KUKA KRL program: Fork_00_Milling_1.src

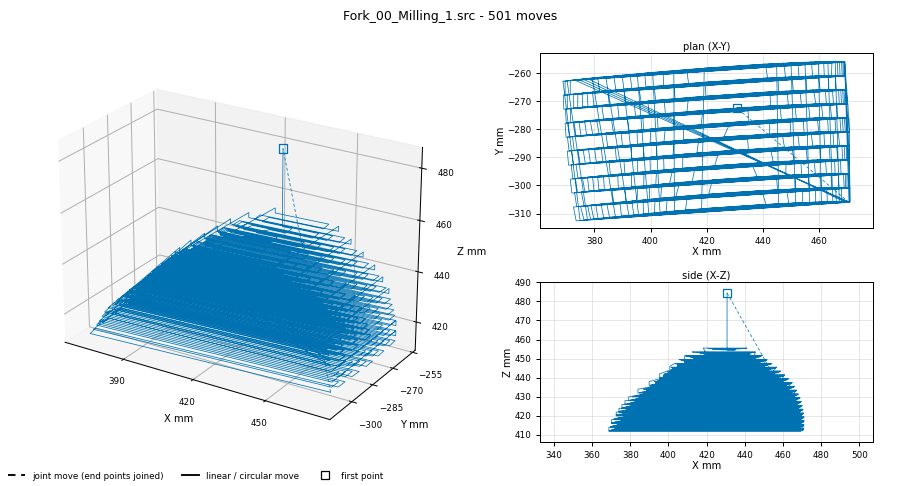
[picture p0: tool path of Fork_00_Milling_1.src, 501 of 503 moves have a stored position in this frame; points joined in program order, loops and branches not executed]
&ACCESS RVP
&REL 1
&PARAM TEMPLATE = C:\KRC\Roboter\Template\vorgabe
&PARAM EDITMASK = *
DEF milling_1 ( )


;FOLD INI
;FOLD BASISTECH INI
GLOBAL INTERRUPT DECL 3 WHEN $STOPMESS==TRUE DO IR_STOPM ( )
INTERRUPT ON 3
BAS (#INITMOV,0 )
;ENDFOLD (BASISTECH INI)
;ENDFOLD (INI)

;FOLD STARTPOSITION - BASE IS 0, TOOL IS 5, SPEED IS 15%, POSITION IS A1 5,A2 -90,A3 100,A4 5,A5 -10,A6 -5,E1 0,E2 0,E3 0,E4 0
$BWDSTART = FALSE
PDAT_ACT = {VEL 15,ACC 100,APO_DIST 50}
FDAT_ACT = {TOOL_NO 5,BASE_NO 0,IPO_FRAME #BASE}
BAS (#PTP_PARAMS,15)
PTP  {A1 5,A2 -90,A3 100,A4 5,A5 -10,A6 -5,E1 0,E2 0,E3 0,E4 0}
;ENDFOLD

;FOLD LIN SPEED IS 0.1 m/sec, INTERPOLATION SETTINGS IN FOLD
$VEL.CP=0.1
$ADVANCE=3
;ENDFOLD

BAS(#VEL_PTP,2)
PTP {X 430.72, Y -272.354, Z 484.436, A 0, B 90, C 0, E1 0, E2 0, E3 0, E4 0, S 'B010'}
$VEL.CP=0.005
LIN {X 430.72, Y -272.354, Z 454.436, A 0, B 90, C 0, E1 0, E2 0, E3 0, E4 0}
LIN {X 434.594, Y -272.091, Z 454.436, A 0, B 90, C 0, E1 0, E2 0, E3 0, E4 0}
LIN {X 435.068, Y -277.068, Z 454.593, A 0, B 90, C 0, E1 0, E2 0, E3 0, E4 0}
LIN {X 428.455, Y -277.517, Z 454.593, A 0, B 90, C 0, E1 0, E2 0, E3 0, E4 0}
LIN {X 426.127, Y -282.684, Z 454.749, A 0, B 90, C 0, E1 0, E2 0, E3 0, E4 0}
LIN {X 434.47, Y -282.118, Z 454.75, A 0, B 90, C 0, E1 0, E2 0, E3 0, E4 0}
LIN {X 434.889, Y -287.099, Z 454.906, A 0, B 90, C 0, E1 0, E2 0, E3 0, E4 0}
LIN {X 424.389, Y -287.811, Z 454.906, A 0, B 90, C 0, E1 0, E2 0, E3 0, E4 0}
LIN {X 422.898, Y -292.921, Z 455.063, A 0, B 90, C 0, E1 0, E2 0, E3 0, E4 0}
LIN {X 435.962, Y -292.035, Z 455.063, A 0, B 90, C 0, E1 0, E2 0, E3 0, E4 0}
LIN {X 437.991, Y -296.906, Z 455.22, A 0, B 90, C 0, E1 0, E2 0, E3 0, E4 0}
LIN {X 422.043, Y -297.989, Z 455.22, A 0, B 90, C 0, E1 0, E2 0, E3 0, E4 0}
LIN {X 420.746, Y -303.086, Z 455.376, A 0, B 90, C 0, E1 0, E2 0, E3 0, E4 0}
LIN {X 439.68, Y -301.801, Z 455.377, A 0, B 90, C 0, E1 0, E2 0, E3 0, E4 0}
LIN {X 441.144, Y -306.71, Z 455.534, A 0, B 90, C 0, E1 0, E2 0, E3 0, E4 0}
LIN {X 418.215, Y -308.266, Z 455.533, A 0, B 90, C 0, E1 0, E2 0, E3 0, E4 0}
LIN {X 419.146, Y -258.113, Z 453.965, A 0, B 90, C 0, E1 0, E2 0, E3 0, E4 0}
LIN {X 419.15, Y -258.175, Z 451.966, A 0, B 90, C 0, E1 0, E2 0, E3 0, E4 0}
LIN {X 440.969, Y -256.694, Z 451.966, A 0, B 90, C 0, E1 0, E2 0, E3 0, E4 0}
LIN {X 441.697, Y -261.654, Z 452.123, A 0, B 90, C 0, E1 0, E2 0, E3 0, E4 0}
LIN {X 419.492, Y -263.161, Z 452.123, A 0, B 90, C 0, E1 0, E2 0, E3 0, E4 0}
LIN {X 419.733, Y -268.154, Z 452.279, A 0, B 90, C 0, E1 0, E2 0, E3 0, E4 0}
LIN {X 442.505, Y -266.608, Z 452.28, A 0, B 90, C 0, E1 0, E2 0, E3 0, E4 0}
LIN {X 442.855, Y -271.594, Z 452.437, A 0, B 90, C 0, E1 0, E2 0, E3 0, E4 0}
LIN {X 418.625, Y -273.238, Z 452.436, A 0, B 90, C 0, E1 0, E2 0, E3 0, E4 0}
LIN {X 418.028, Y -278.288, Z 452.593, A 0, B 90, C 0, E1 0, E2 0, E3 0, E4 0}
LIN {X 442.441, Y -276.631, Z 452.594, A 0, B 90, C 0, E1 0, E2 0, E3 0, E4 0}
LIN {X 442.487, Y -281.637, Z 452.75, A 0, B 90, C 0, E1 0, E2 0, E3 0, E4 0}
LIN {X 417.259, Y -283.349, Z 452.75, A 0, B 90, C 0, E1 0, E2 0, E3 0, E4 0}
LIN {X 416.509, Y -288.409, Z 452.906, A 0, B 90, C 0, E1 0, E2 0, E3 0, E4 0}
LIN {X 442.672, Y -286.633, Z 452.907, A 0, B 90, C 0, E1 0, E2 0, E3 0, E4 0}
LIN {X 443.761, Y -291.568, Z 453.064, A 0, B 90, C 0, E1 0, E2 0, E3 0, E4 0}
LIN {X 415.871, Y -293.461, Z 453.063, A 0, B 90, C 0, E1 0, E2 0, E3 0, E4 0}
LIN {X 414.841, Y -298.54, Z 453.22, A 0, B 90, C 0, E1 0, E2 0, E3 0, E4 0}
LIN {X 444.838, Y -296.504, Z 453.221, A 0, B 90, C 0, E1 0, E2 0, E3 0, E4 0}
LIN {X 445.27, Y -301.484, Z 453.378, A 0, B 90, C 0, E1 0, E2 0, E3 0, E4 0}
LIN {X 413.14, Y -303.665, Z 453.377, A 0, B 90, C 0, E1 0, E2 0, E3 0, E4 0}
LIN {X 412.448, Y -308.721, Z 453.534, A 0, B 90, C 0, E1 0, E2 0, E3 0, E4 0}
LIN {X 445.669, Y -306.466, Z 453.534, A 0, B 90, C 0, E1 0, E2 0, E3 0, E4 0}
LIN {X 444.959, Y -256.424, Z 451.967, A 0, B 90, C 0, E1 0, E2 0, E3 0, E4 0}
LIN {X 444.964, Y -256.486, Z 449.968, A 0, B 90, C 0, E1 0, E2 0, E3 0, E4 0}
LIN {X 412.911, Y -258.662, Z 449.967, A 0, B 90, C 0, E1 0, E2 0, E3 0, E4 0}
LIN {X 413.546, Y -263.628, Z 450.124, A 0, B 90, C 0, E1 0, E2 0, E3 0, E4 0}
LIN {X 445.401, Y -261.466, Z 450.124, A 0, B 90, C 0, E1 0, E2 0, E3 0, E4 0}
LIN {X 445.696, Y -266.455, Z 450.281, A 0, B 90, C 0, E1 0, E2 0, E3 0, E4 0}
LIN {X 413.503, Y -268.64, Z 450.281, A 0, B 90, C 0, E1 0, E2 0, E3 0, E4 0}
LIN {X 413.007, Y -273.682, Z 450.437, A 0, B 90, C 0, E1 0, E2 0, E3 0, E4 0}
LIN {X 446.106, Y -271.436, Z 450.438, A 0, B 90, C 0, E1 0, E2 0, E3 0, E4 0}
LIN {X 446.657, Y -276.407, Z 450.595, A 0, B 90, C 0, E1 0, E2 0, E3 0, E4 0}
LIN {X 411.832, Y -278.771, Z 450.594, A 0, B 90, C 0, E1 0, E2 0, E3 0, E4 0}
LIN {X 411.67, Y -283.791, Z 450.751, A 0, B 90, C 0, E1 0, E2 0, E3 0, E4 0}
LIN {X 446.887, Y -281.401, Z 450.752, A 0, B 90, C 0, E1 0, E2 0, E3 0, E4 0}
LIN {X 447.736, Y -286.352, Z 450.908, A 0, B 90, C 0, E1 0, E2 0, E3 0, E4 0}
LIN {X 411.519, Y -288.811, Z 450.908, A 0, B 90, C 0, E1 0, E2 0, E3 0, E4 0}
LIN {X 411.454, Y -293.824, Z 451.064, A 0, B 90, C 0, E1 0, E2 0, E3 0, E4 0}
LIN {X 448.317, Y -291.322, Z 451.065, A 0, B 90, C 0, E1 0, E2 0, E3 0, E4 0}
LIN {X 448.215, Y -296.338, Z 451.222, A 0, B 90, C 0, E1 0, E2 0, E3 0, E4 0}
LIN {X 410.374, Y -298.906, Z 451.221, A 0, B 90, C 0, E1 0, E2 0, E3 0, E4 0}
LIN {X 409.012, Y -304.008, Z 451.378, A 0, B 90, C 0, E1 0, E2 0, E3 0, E4 0}
LIN {X 448.504, Y -301.327, Z 451.379, A 0, B 90, C 0, E1 0, E2 0, E3 0, E4 0}
LIN {X 449.256, Y -306.285, Z 451.536, A 0, B 90, C 0, E1 0, E2 0, E3 0, E4 0}
LIN {X 408.508, Y -309.051, Z 451.535, A 0, B 90, C 0, E1 0, E2 0, E3 0, E4 0}
LIN {X 408.295, Y -258.975, Z 449.967, A 0, B 90, C 0, E1 0, E2 0, E3 0, E4 0}
LIN {X 408.299, Y -259.038, Z 447.968, A 0, B 90, C 0, E1 0, E2 0, E3 0, E4 0}
LIN {X 447.536, Y -256.374, Z 447.969, A 0, B 90, C 0, E1 0, E2 0, E3 0, E4 0}
LIN {X 448.106, Y -261.345, Z 448.126, A 0, B 90, C 0, E1 0, E2 0, E3 0, E4 0}
LIN {X 408.404, Y -264.04, Z 448.125, A 0, B 90, C 0, E1 0, E2 0, E3 0, E4 0}
LIN {X 408.727, Y -269.027, Z 448.281, A 0, B 90, C 0, E1 0, E2 0, E3 0, E4 0}
LIN {X 448.61, Y -266.32, Z 448.282, A 0, B 90, C 0, E1 0, E2 0, E3 0, E4 0}
LIN {X 449.134, Y -271.293, Z 448.439, A 0, B 90, C 0, E1 0, E2 0, E3 0, E4 0}
LIN {X 408.355, Y -274.061, Z 448.438, A 0, B 90, C 0, E1 0, E2 0, E3 0, E4 0}
LIN {X 408.359, Y -279.07, Z 448.595, A 0, B 90, C 0, E1 0, E2 0, E3 0, E4 0}
LIN {X 449.68, Y -276.265, Z 448.596, A 0, B 90, C 0, E1 0, E2 0, E3 0, E4 0}
LIN {X 450.001, Y -281.252, Z 448.753, A 0, B 90, C 0, E1 0, E2 0, E3 0, E4 0}
LIN {X 408.293, Y -284.083, Z 448.752, A 0, B 90, C 0, E1 0, E2 0, E3 0, E4 0}
LIN {X 408.039, Y -289.11, Z 448.909, A 0, B 90, C 0, E1 0, E2 0, E3 0, E4 0}
LIN {X 450.372, Y -286.236, Z 448.909, A 0, B 90, C 0, E1 0, E2 0, E3 0, E4 0}
LIN {X 451.141, Y -291.193, Z 449.066, A 0, B 90, C 0, E1 0, E2 0, E3 0, E4 0}
LIN {X 407.934, Y -294.126, Z 449.065, A 0, B 90, C 0, E1 0, E2 0, E3 0, E4 0}
LIN {X 406.788, Y -299.213, Z 449.222, A 0, B 90, C 0, E1 0, E2 0, E3 0, E4 0}
LIN {X 451.562, Y -296.174, Z 449.223, A 0, B 90, C 0, E1 0, E2 0, E3 0, E4 0}
LIN {X 451.599, Y -301.18, Z 449.38, A 0, B 90, C 0, E1 0, E2 0, E3 0, E4 0}
LIN {X 405.979, Y -304.277, Z 449.379, A 0, B 90, C 0, E1 0, E2 0, E3 0, E4 0}
LIN {X 405.553, Y -309.315, Z 449.536, A 0, B 90, C 0, E1 0, E2 0, E3 0, E4 0}
LIN {X 451.726, Y -306.18, Z 449.537, A 0, B 90, C 0, E1 0, E2 0, E3 0, E4 0}
LIN {X 450.067, Y -256.203, Z 447.969, A 0, B 90, C 0, E1 0, E2 0, E3 0, E4 0}
LIN {X 450.071, Y -256.265, Z 445.97, A 0, B 90, C 0, E1 0, E2 0, E3 0, E4 0}
LIN {X 404.497, Y -259.359, Z 445.969, A 0, B 90, C 0, E1 0, E2 0, E3 0, E4 0}
LIN {X 404.613, Y -264.36, Z 446.125, A 0, B 90, C 0, E1 0, E2 0, E3 0, E4 0}
LIN {X 450.414, Y -261.251, Z 446.127, A 0, B 90, C 0, E1 0, E2 0, E3 0, E4 0}
LIN {X 450.904, Y -266.227, Z 446.283, A 0, B 90, C 0, E1 0, E2 0, E3 0, E4 0}
LIN {X 404.855, Y -269.352, Z 446.282, A 0, B 90, C 0, E1 0, E2 0, E3 0, E4 0}
LIN {X 405.282, Y -274.333, Z 446.439, A 0, B 90, C 0, E1 0, E2 0, E3 0, E4 0}
LIN {X 451.426, Y -271.2, Z 446.44, A 0, B 90, C 0, E1 0, E2 0, E3 0, E4 0}
LIN {X 451.972, Y -276.172, Z 446.597, A 0, B 90, C 0, E1 0, E2 0, E3 0, E4 0}
LIN {X 405.292, Y -279.341, Z 446.596, A 0, B 90, C 0, E1 0, E2 0, E3 0, E4 0}
LIN {X 404.784, Y -284.384, Z 446.753, A 0, B 90, C 0, E1 0, E2 0, E3 0, E4 0}
LIN {X 452.413, Y -281.151, Z 446.754, A 0, B 90, C 0, E1 0, E2 0, E3 0, E4 0}
LIN {X 453.043, Y -286.118, Z 446.911, A 0, B 90, C 0, E1 0, E2 0, E3 0, E4 0}
LIN {X 404.634, Y -289.404, Z 446.909, A 0, B 90, C 0, E1 0, E2 0, E3 0, E4 0}
LIN {X 404.807, Y -294.401, Z 447.066, A 0, B 90, C 0, E1 0, E2 0, E3 0, E4 0}
LIN {X 453.573, Y -291.091, Z 447.067, A 0, B 90, C 0, E1 0, E2 0, E3 0, E4 0}
LIN {X 453.857, Y -296.081, Z 447.224, A 0, B 90, C 0, E1 0, E2 0, E3 0, E4 0}
LIN {X 404.012, Y -299.464, Z 447.223, A 0, B 90, C 0, E1 0, E2 0, E3 0, E4 0}
LIN {X 403.621, Y -304.499, Z 447.38, A 0, B 90, C 0, E1 0, E2 0, E3 0, E4 0}
LIN {X 454.257, Y -301.063, Z 447.381, A 0, B 90, C 0, E1 0, E2 0, E3 0, E4 0}
LIN {X 454.181, Y -306.077, Z 447.538, A 0, B 90, C 0, E1 0, E2 0, E3 0, E4 0}
LIN {X 403.378, Y -309.525, Z 447.536, A 0, B 90, C 0, E1 0, E2 0, E3 0, E4 0}
LIN {X 400.738, Y -259.614, Z 445.969, A 0, B 90, C 0, E1 0, E2 0, E3 0, E4 0}
LIN {X 400.743, Y -259.676, Z 443.969, A 0, B 90, C 0, E1 0, E2 0, E3 0, E4 0}
LIN {X 452.557, Y -256.159, Z 443.971, A 0, B 90, C 0, E1 0, E2 0, E3 0, E4 0}
LIN {X 452.9, Y -261.145, Z 444.127, A 0, B 90, C 0, E1 0, E2 0, E3 0, E4 0}
LIN {X 401.269, Y -264.65, Z 444.126, A 0, B 90, C 0, E1 0, E2 0, E3 0, E4 0}
LIN {X 401.82, Y -269.621, Z 444.283, A 0, B 90, C 0, E1 0, E2 0, E3 0, E4 0}
LIN {X 453.243, Y -266.131, Z 444.284, A 0, B 90, C 0, E1 0, E2 0, E3 0, E4 0}
LIN {X 453.757, Y -271.105, Z 444.441, A 0, B 90, C 0, E1 0, E2 0, E3 0, E4 0}
LIN {X 402.363, Y -274.594, Z 444.44, A 0, B 90, C 0, E1 0, E2 0, E3 0, E4 0}
LIN {X 402.668, Y -279.582, Z 444.597, A 0, B 90, C 0, E1 0, E2 0, E3 0, E4 0}
LIN {X 454.371, Y -276.072, Z 444.598, A 0, B 90, C 0, E1 0, E2 0, E3 0, E4 0}
LIN {X 454.728, Y -281.057, Z 444.755, A 0, B 90, C 0, E1 0, E2 0, E3 0, E4 0}
LIN {X 402.155, Y -284.626, Z 444.753, A 0, B 90, C 0, E1 0, E2 0, E3 0, E4 0}
LIN {X 402.095, Y -289.639, Z 444.91, A 0, B 90, C 0, E1 0, E2 0, E3 0, E4 0}
LIN {X 455.371, Y -286.023, Z 444.911, A 0, B 90, C 0, E1 0, E2 0, E3 0, E4 0}
LIN {X 455.856, Y -290.999, Z 445.068, A 0, B 90, C 0, E1 0, E2 0, E3 0, E4 0}
LIN {X 402.122, Y -294.646, Z 445.067, A 0, B 90, C 0, E1 0, E2 0, E3 0, E4 0}
LIN {X 401.877, Y -299.672, Z 445.224, A 0, B 90, C 0, E1 0, E2 0, E3 0, E4 0}
LIN {X 456.278, Y -295.979, Z 445.225, A 0, B 90, C 0, E1 0, E2 0, E3 0, E4 0}
LIN {X 456.604, Y -300.966, Z 445.382, A 0, B 90, C 0, E1 0, E2 0, E3 0, E4 0}
LIN {X 401.627, Y -304.698, Z 445.381, A 0, B 90, C 0, E1 0, E2 0, E3 0, E4 0}
LIN {X 401.381, Y -309.723, Z 445.537, A 0, B 90, C 0, E1 0, E2 0, E3 0, E4 0}
LIN {X 456.676, Y -305.97, Z 445.539, A 0, B 90, C 0, E1 0, E2 0, E3 0, E4 0}
LIN {X 455.057, Y -255.99, Z 443.971, A 0, B 90, C 0, E1 0, E2 0, E3 0, E4 0}
LIN {X 455.062, Y -256.052, Z 441.972, A 0, B 90, C 0, E1 0, E2 0, E3 0, E4 0}
LIN {X 397.907, Y -259.932, Z 441.97, A 0, B 90, C 0, E1 0, E2 0, E3 0, E4 0}
LIN {X 398.366, Y -264.91, Z 442.127, A 0, B 90, C 0, E1 0, E2 0, E3 0, E4 0}
LIN {X 455.403, Y -261.038, Z 442.128, A 0, B 90, C 0, E1 0, E2 0, E3 0, E4 0}
LIN {X 455.72, Y -266.026, Z 442.285, A 0, B 90, C 0, E1 0, E2 0, E3 0, E4 0}
LIN {X 398.99, Y -269.876, Z 442.284, A 0, B 90, C 0, E1 0, E2 0, E3 0, E4 0}
LIN {X 399.564, Y -274.846, Z 442.441, A 0, B 90, C 0, E1 0, E2 0, E3 0, E4 0}
LIN {X 456.275, Y -270.997, Z 442.442, A 0, B 90, C 0, E1 0, E2 0, E3 0, E4 0}
LIN {X 456.818, Y -275.969, Z 442.599, A 0, B 90, C 0, E1 0, E2 0, E3 0, E4 0}
LIN {X 400.065, Y -279.821, Z 442.597, A 0, B 90, C 0, E1 0, E2 0, E3 0, E4 0}
LIN {X 399.84, Y -284.846, Z 442.754, A 0, B 90, C 0, E1 0, E2 0, E3 0, E4 0}
LIN {X 457.204, Y -280.952, Z 442.756, A 0, B 90, C 0, E1 0, E2 0, E3 0, E4 0}
LIN {X 457.852, Y -285.917, Z 442.912, A 0, B 90, C 0, E1 0, E2 0, E3 0, E4 0}
LIN {X 399.811, Y -289.857, Z 442.911, A 0, B 90, C 0, E1 0, E2 0, E3 0, E4 0}
LIN {X 399.908, Y -294.859, Z 443.068, A 0, B 90, C 0, E1 0, E2 0, E3 0, E4 0}
LIN {X 458.35, Y -290.892, Z 443.069, A 0, B 90, C 0, E1 0, E2 0, E3 0, E4 0}
LIN {X 458.732, Y -295.875, Z 443.226, A 0, B 90, C 0, E1 0, E2 0, E3 0, E4 0}
LIN {X 399.751, Y -299.879, Z 443.225, A 0, B 90, C 0, E1 0, E2 0, E3 0, E4 0}
LIN {X 399.552, Y -304.901, Z 443.381, A 0, B 90, C 0, E1 0, E2 0, E3 0, E4 0}
LIN {X 458.809, Y -300.879, Z 443.383, A 0, B 90, C 0, E1 0, E2 0, E3 0, E4 0}
LIN {X 458.885, Y -305.883, Z 443.54, A 0, B 90, C 0, E1 0, E2 0, E3 0, E4 0}
LIN {X 399.354, Y -309.924, Z 443.538, A 0, B 90, C 0, E1 0, E2 0, E3 0, E4 0}
LIN {X 395.258, Y -260.112, Z 441.97, A 0, B 90, C 0, E1 0, E2 0, E3 0, E4 0}
LIN {X 395.262, Y -260.174, Z 439.971, A 0, B 90, C 0, E1 0, E2 0, E3 0, E4 0}
LIN {X 457.344, Y -255.96, Z 439.972, A 0, B 90, C 0, E1 0, E2 0, E3 0, E4 0}
LIN {X 457.776, Y -260.94, Z 440.129, A 0, B 90, C 0, E1 0, E2 0, E3 0, E4 0}
LIN {X 395.84, Y -265.144, Z 440.128, A 0, B 90, C 0, E1 0, E2 0, E3 0, E4 0}
LIN {X 396.614, Y -270.1, Z 440.285, A 0, B 90, C 0, E1 0, E2 0, E3 0, E4 0}
LIN {X 458.111, Y -265.926, Z 440.286, A 0, B 90, C 0, E1 0, E2 0, E3 0, E4 0}
LIN {X 458.91, Y -270.881, Z 440.443, A 0, B 90, C 0, E1 0, E2 0, E3 0, E4 0}
LIN {X 397.252, Y -275.066, Z 440.441, A 0, B 90, C 0, E1 0, E2 0, E3 0, E4 0}
LIN {X 397.475, Y -280.06, Z 440.598, A 0, B 90, C 0, E1 0, E2 0, E3 0, E4 0}
LIN {X 459.417, Y -275.856, Z 440.6, A 0, B 90, C 0, E1 0, E2 0, E3 0, E4 0}
LIN {X 459.985, Y -280.826, Z 440.756, A 0, B 90, C 0, E1 0, E2 0, E3 0, E4 0}
LIN {X 397.521, Y -285.066, Z 440.755, A 0, B 90, C 0, E1 0, E2 0, E3 0, E4 0}
LIN {X 397.583, Y -290.071, Z 440.912, A 0, B 90, C 0, E1 0, E2 0, E3 0, E4 0}
LIN {X 460.359, Y -285.81, Z 440.913, A 0, B 90, C 0, E1 0, E2 0, E3 0, E4 0}
LIN {X 460.544, Y -290.806, Z 441.07, A 0, B 90, C 0, E1 0, E2 0, E3 0, E4 0}
LIN {X 397.674, Y -295.074, Z 441.069, A 0, B 90, C 0, E1 0, E2 0, E3 0, E4 0}
LIN {X 397.572, Y -300.09, Z 441.225, A 0, B 90, C 0, E1 0, E2 0, E3 0, E4 0}
LIN {X 460.729, Y -295.803, Z 441.227, A 0, B 90, C 0, E1 0, E2 0, E3 0, E4 0}
LIN {X 460.84, Y -300.804, Z 441.384, A 0, B 90, C 0, E1 0, E2 0, E3 0, E4 0}
LIN {X 397.374, Y -305.112, Z 441.382, A 0, B 90, C 0, E1 0, E2 0, E3 0, E4 0}
LIN {X 397.441, Y -310.117, Z 441.539, A 0, B 90, C 0, E1 0, E2 0, E3 0, E4 0}
LIN {X 460.897, Y -305.809, Z 441.54, A 0, B 90, C 0, E1 0, E2 0, E3 0, E4 0}
LIN {X 459.838, Y -255.791, Z 439.972, A 0, B 90, C 0, E1 0, E2 0, E3 0, E4 0}
LIN {X 459.842, Y -255.853, Z 437.973, A 0, B 90, C 0, E1 0, E2 0, E3 0, E4 0}
LIN {X 392.711, Y -260.41, Z 437.972, A 0, B 90, C 0, E1 0, E2 0, E3 0, E4 0}
LIN {X 393.304, Y -265.379, Z 438.129, A 0, B 90, C 0, E1 0, E2 0, E3 0, E4 0}
LIN {X 459.891, Y -260.859, Z 438.13, A 0, B 90, C 0, E1 0, E2 0, E3 0, E4 0}
LIN {X 460.475, Y -265.829, Z 438.287, A 0, B 90, C 0, E1 0, E2 0, E3 0, E4 0}
LIN {X 394.093, Y -270.334, Z 438.285, A 0, B 90, C 0, E1 0, E2 0, E3 0, E4 0}
LIN {X 394.69, Y -275.303, Z 438.442, A 0, B 90, C 0, E1 0, E2 0, E3 0, E4 0}
LIN {X 460.924, Y -270.807, Z 438.444, A 0, B 90, C 0, E1 0, E2 0, E3 0, E4 0}
LIN {X 461.398, Y -275.784, Z 438.601, A 0, B 90, C 0, E1 0, E2 0, E3 0, E4 0}
LIN {X 395.156, Y -280.28, Z 438.599, A 0, B 90, C 0, E1 0, E2 0, E3 0, E4 0}
LIN {X 395.334, Y -285.277, Z 438.756, A 0, B 90, C 0, E1 0, E2 0, E3 0, E4 0}
LIN {X 461.793, Y -280.766, Z 438.757, A 0, B 90, C 0, E1 0, E2 0, E3 0, E4 0}
LIN {X 462.025, Y -285.76, Z 438.914, A 0, B 90, C 0, E1 0, E2 0, E3 0, E4 0}
LIN {X 395.356, Y -290.285, Z 438.913, A 0, B 90, C 0, E1 0, E2 0, E3 0, E4 0}
LIN {X 395.431, Y -295.289, Z 439.069, A 0, B 90, C 0, E1 0, E2 0, E3 0, E4 0}
LIN {X 462.369, Y -290.745, Z 439.071, A 0, B 90, C 0, E1 0, E2 0, E3 0, E4 0}
LIN {X 462.701, Y -295.732, Z 439.228, A 0, B 90, C 0, E1 0, E2 0, E3 0, E4 0}
LIN {X 395.383, Y -300.301, Z 439.226, A 0, B 90, C 0, E1 0, E2 0, E3 0, E4 0}
LIN {X 395.185, Y -305.324, Z 439.383, A 0, B 90, C 0, E1 0, E2 0, E3 0, E4 0}
LIN {X 462.857, Y -300.73, Z 439.384, A 0, B 90, C 0, E1 0, E2 0, E3 0, E4 0}
LIN {X 463.008, Y -305.729, Z 439.541, A 0, B 90, C 0, E1 0, E2 0, E3 0, E4 0}
LIN {X 395.705, Y -310.297, Z 439.54, A 0, B 90, C 0, E1 0, E2 0, E3 0, E4 0}
LIN {X 389.875, Y -260.603, Z 437.972, A 0, B 90, C 0, E1 0, E2 0, E3 0, E4 0}
LIN {X 389.879, Y -260.665, Z 435.973, A 0, B 90, C 0, E1 0, E2 0, E3 0, E4 0}
LIN {X 461.709, Y -255.79, Z 435.974, A 0, B 90, C 0, E1 0, E2 0, E3 0, E4 0}
LIN {X 461.933, Y -260.783, Z 436.131, A 0, B 90, C 0, E1 0, E2 0, E3 0, E4 0}
LIN {X 390.561, Y -265.628, Z 436.129, A 0, B 90, C 0, E1 0, E2 0, E3 0, E4 0}
LIN {X 391.138, Y -270.598, Z 436.286, A 0, B 90, C 0, E1 0, E2 0, E3 0, E4 0}
LIN {X 462.277, Y -265.769, Z 436.288, A 0, B 90, C 0, E1 0, E2 0, E3 0, E4 0}
LIN {X 462.678, Y -270.751, Z 436.445, A 0, B 90, C 0, E1 0, E2 0, E3 0, E4 0}
LIN {X 391.714, Y -275.568, Z 436.443, A 0, B 90, C 0, E1 0, E2 0, E3 0, E4 0}
LIN {X 392.348, Y -280.534, Z 436.6, A 0, B 90, C 0, E1 0, E2 0, E3 0, E4 0}
LIN {X 463.08, Y -275.733, Z 436.602, A 0, B 90, C 0, E1 0, E2 0, E3 0, E4 0}
LIN {X 463.38, Y -280.721, Z 436.758, A 0, B 90, C 0, E1 0, E2 0, E3 0, E4 0}
LIN {X 393.096, Y -285.492, Z 436.757, A 0, B 90, C 0, E1 0, E2 0, E3 0, E4 0}
LIN {X 393.301, Y -290.487, Z 436.913, A 0, B 90, C 0, E1 0, E2 0, E3 0, E4 0}
LIN {X 463.651, Y -285.712, Z 436.915, A 0, B 90, C 0, E1 0, E2 0, E3 0, E4 0}
LIN {X 463.996, Y -290.698, Z 437.072, A 0, B 90, C 0, E1 0, E2 0, E3 0, E4 0}
LIN {X 393.202, Y -295.503, Z 437.07, A 0, B 90, C 0, E1 0, E2 0, E3 0, E4 0}
LIN {X 393.16, Y -300.515, Z 437.227, A 0, B 90, C 0, E1 0, E2 0, E3 0, E4 0}
LIN {X 464.339, Y -295.683, Z 437.229, A 0, B 90, C 0, E1 0, E2 0, E3 0, E4 0}
LIN {X 464.542, Y -300.679, Z 437.385, A 0, B 90, C 0, E1 0, E2 0, E3 0, E4 0}
LIN {X 393.32, Y -305.513, Z 437.384, A 0, B 90, C 0, E1 0, E2 0, E3 0, E4 0}
LIN {X 394.013, Y -310.475, Z 437.541, A 0, B 90, C 0, E1 0, E2 0, E3 0, E4 0}
LIN {X 464.996, Y -305.657, Z 437.542, A 0, B 90, C 0, E1 0, E2 0, E3 0, E4 0}
LIN {X 463.196, Y -255.689, Z 435.974, A 0, B 90, C 0, E1 0, E2 0, E3 0, E4 0}
LIN {X 463.2, Y -255.751, Z 433.975, A 0, B 90, C 0, E1 0, E2 0, E3 0, E4 0}
LIN {X 386.906, Y -260.93, Z 433.974, A 0, B 90, C 0, E1 0, E2 0, E3 0, E4 0}
LIN {X 387.629, Y -265.89, Z 434.13, A 0, B 90, C 0, E1 0, E2 0, E3 0, E4 0}
LIN {X 463.279, Y -260.755, Z 434.132, A 0, B 90, C 0, E1 0, E2 0, E3 0, E4 0}
LIN {X 463.532, Y -265.747, Z 434.289, A 0, B 90, C 0, E1 0, E2 0, E3 0, E4 0}
LIN {X 388.206, Y -270.86, Z 434.287, A 0, B 90, C 0, E1 0, E2 0, E3 0, E4 0}
LIN {X 388.783, Y -275.83, Z 434.444, A 0, B 90, C 0, E1 0, E2 0, E3 0, E4 0}
LIN {X 464.021, Y -270.723, Z 434.446, A 0, B 90, C 0, E1 0, E2 0, E3 0, E4 0}
LIN {X 464.51, Y -275.699, Z 434.602, A 0, B 90, C 0, E1 0, E2 0, E3 0, E4 0}
LIN {X 389.454, Y -280.793, Z 434.601, A 0, B 90, C 0, E1 0, E2 0, E3 0, E4 0}
LIN {X 389.986, Y -285.766, Z 434.758, A 0, B 90, C 0, E1 0, E2 0, E3 0, E4 0}
LIN {X 464.983, Y -280.675, Z 434.759, A 0, B 90, C 0, E1 0, E2 0, E3 0, E4 0}
LIN {X 465.324, Y -285.661, Z 434.916, A 0, B 90, C 0, E1 0, E2 0, E3 0, E4 0}
LIN {X 390.481, Y -290.741, Z 434.914, A 0, B 90, C 0, E1 0, E2 0, E3 0, E4 0}
LIN {X 390.853, Y -295.725, Z 435.071, A 0, B 90, C 0, E1 0, E2 0, E3 0, E4 0}
LIN {X 465.594, Y -290.652, Z 435.073, A 0, B 90, C 0, E1 0, E2 0, E3 0, E4 0}
LIN {X 465.794, Y -295.648, Z 435.23, A 0, B 90, C 0, E1 0, E2 0, E3 0, E4 0}
LIN {X 390.798, Y -300.738, Z 435.228, A 0, B 90, C 0, E1 0, E2 0, E3 0, E4 0}
LIN {X 391.209, Y -305.719, Z 435.385, A 0, B 90, C 0, E1 0, E2 0, E3 0, E4 0}
LIN {X 465.993, Y -300.643, Z 435.386, A 0, B 90, C 0, E1 0, E2 0, E3 0, E4 0}
LIN {X 466.217, Y -305.637, Z 435.543, A 0, B 90, C 0, E1 0, E2 0, E3 0, E4 0}
LIN {X 392.262, Y -310.657, Z 435.541, A 0, B 90, C 0, E1 0, E2 0, E3 0, E4 0}
LIN {X 384.003, Y -261.127, Z 433.973, A 0, B 90, C 0, E1 0, E2 0, E3 0, E4 0}
LIN {X 384.007, Y -261.189, Z 431.974, A 0, B 90, C 0, E1 0, E2 0, E3 0, E4 0}
LIN {X 464.665, Y -255.715, Z 431.976, A 0, B 90, C 0, E1 0, E2 0, E3 0, E4 0}
LIN {X 464.52, Y -260.734, Z 432.133, A 0, B 90, C 0, E1 0, E2 0, E3 0, E4 0}
LIN {X 384.71, Y -266.151, Z 432.131, A 0, B 90, C 0, E1 0, E2 0, E3 0, E4 0}
LIN {X 385.287, Y -271.121, Z 432.288, A 0, B 90, C 0, E1 0, E2 0, E3 0, E4 0}
LIN {X 464.818, Y -265.722, Z 432.29, A 0, B 90, C 0, E1 0, E2 0, E3 0, E4 0}
LIN {X 465.216, Y -270.704, Z 432.447, A 0, B 90, C 0, E1 0, E2 0, E3 0, E4 0}
LIN {X 386.03, Y -276.079, Z 432.445, A 0, B 90, C 0, E1 0, E2 0, E3 0, E4 0}
LIN {X 386.741, Y -281.04, Z 432.601, A 0, B 90, C 0, E1 0, E2 0, E3 0, E4 0}
LIN {X 465.705, Y -275.68, Z 432.603, A 0, B 90, C 0, E1 0, E2 0, E3 0, E4 0}
LIN {X 466.049, Y -280.666, Z 432.76, A 0, B 90, C 0, E1 0, E2 0, E3 0, E4 0}
LIN {X 387.361, Y -286.007, Z 432.758, A 0, B 90, C 0, E1 0, E2 0, E3 0, E4 0}
LIN {X 387.839, Y -290.984, Z 432.915, A 0, B 90, C 0, E1 0, E2 0, E3 0, E4 0}
LIN {X 466.305, Y -285.658, Z 432.917, A 0, B 90, C 0, E1 0, E2 0, E3 0, E4 0}
LIN {X 466.702, Y -290.64, Z 433.074, A 0, B 90, C 0, E1 0, E2 0, E3 0, E4 0}
LIN {X 388.304, Y -295.961, Z 433.072, A 0, B 90, C 0, E1 0, E2 0, E3 0, E4 0}
LIN {X 388.51, Y -300.956, Z 433.229, A 0, B 90, C 0, E1 0, E2 0, E3 0, E4 0}
LIN {X 466.934, Y -295.633, Z 433.23, A 0, B 90, C 0, E1 0, E2 0, E3 0, E4 0}
LIN {X 467.135, Y -300.628, Z 433.387, A 0, B 90, C 0, E1 0, E2 0, E3 0, E4 0}
LIN {X 389.063, Y -305.928, Z 433.385, A 0, B 90, C 0, E1 0, E2 0, E3 0, E4 0}
LIN {X 389.632, Y -310.898, Z 433.542, A 0, B 90, C 0, E1 0, E2 0, E3 0, E4 0}
LIN {X 467.285, Y -305.627, Z 433.544, A 0, B 90, C 0, E1 0, E2 0, E3 0, E4 0}
LIN {X 465.823, Y -255.636, Z 431.976, A 0, B 90, C 0, E1 0, E2 0, E3 0, E4 0}
LIN {X 465.827, Y -255.699, Z 429.977, A 0, B 90, C 0, E1 0, E2 0, E3 0, E4 0}
LIN {X 381.164, Y -261.445, Z 429.975, A 0, B 90, C 0, E1 0, E2 0, E3 0, E4 0}
LIN {X 381.818, Y -266.41, Z 430.132, A 0, B 90, C 0, E1 0, E2 0, E3 0, E4 0}
LIN {X 465.818, Y -260.708, Z 430.134, A 0, B 90, C 0, E1 0, E2 0, E3 0, E4 0}
LIN {X 466.116, Y -265.697, Z 430.291, A 0, B 90, C 0, E1 0, E2 0, E3 0, E4 0}
LIN {X 382.579, Y -271.367, Z 430.289, A 0, B 90, C 0, E1 0, E2 0, E3 0, E4 0}
LIN {X 383.306, Y -276.327, Z 430.445, A 0, B 90, C 0, E1 0, E2 0, E3 0, E4 0}
LIN {X 466.414, Y -270.686, Z 430.447, A 0, B 90, C 0, E1 0, E2 0, E3 0, E4 0}
LIN {X 466.688, Y -275.676, Z 430.604, A 0, B 90, C 0, E1 0, E2 0, E3 0, E4 0}
LIN {X 384.017, Y -281.288, Z 430.602, A 0, B 90, C 0, E1 0, E2 0, E3 0, E4 0}
LIN {X 384.778, Y -286.245, Z 430.759, A 0, B 90, C 0, E1 0, E2 0, E3 0, E4 0}
LIN {X 466.875, Y -280.673, Z 430.761, A 0, B 90, C 0, E1 0, E2 0, E3 0, E4 0}
LIN {X 467.385, Y -285.647, Z 430.918, A 0, B 90, C 0, E1 0, E2 0, E3 0, E4 0}
LIN {X 385.205, Y -291.225, Z 430.916, A 0, B 90, C 0, E1 0, E2 0, E3 0, E4 0}
LIN {X 385.676, Y -296.202, Z 431.073, A 0, B 90, C 0, E1 0, E2 0, E3 0, E4 0}
LIN {X 467.687, Y -290.636, Z 431.075, A 0, B 90, C 0, E1 0, E2 0, E3 0, E4 0}
LIN {X 467.909, Y -295.63, Z 431.231, A 0, B 90, C 0, E1 0, E2 0, E3 0, E4 0}
LIN {X 386.199, Y -301.176, Z 431.229, A 0, B 90, C 0, E1 0, E2 0, E3 0, E4 0}
LIN {X 386.84, Y -306.141, Z 431.386, A 0, B 90, C 0, E1 0, E2 0, E3 0, E4 0}
LIN {X 468.106, Y -300.625, Z 431.388, A 0, B 90, C 0, E1 0, E2 0, E3 0, E4 0}
LIN {X 468.083, Y -305.636, Z 431.545, A 0, B 90, C 0, E1 0, E2 0, E3 0, E4 0}
LIN {X 387.48, Y -311.107, Z 431.543, A 0, B 90, C 0, E1 0, E2 0, E3 0, E4 0}
LIN {X 379.164, Y -261.581, Z 429.975, A 0, B 90, C 0, E1 0, E2 0, E3 0, E4 0}
LIN {X 379.168, Y -261.644, Z 427.976, A 0, B 90, C 0, E1 0, E2 0, E3 0, E4 0}
LIN {X 466.586, Y -255.71, Z 427.978, A 0, B 90, C 0, E1 0, E2 0, E3 0, E4 0}
LIN {X 466.792, Y -260.705, Z 428.135, A 0, B 90, C 0, E1 0, E2 0, E3 0, E4 0}
LIN {X 379.275, Y -266.645, Z 428.133, A 0, B 90, C 0, E1 0, E2 0, E3 0, E4 0}
LIN {X 379.839, Y -271.616, Z 428.29, A 0, B 90, C 0, E1 0, E2 0, E3 0, E4 0}
LIN {X 467.026, Y -265.698, Z 428.292, A 0, B 90, C 0, E1 0, E2 0, E3 0, E4 0}
LIN {X 467.273, Y -270.691, Z 428.448, A 0, B 90, C 0, E1 0, E2 0, E3 0, E4 0}
LIN {X 380.73, Y -276.565, Z 428.446, A 0, B 90, C 0, E1 0, E2 0, E3 0, E4 0}
LIN {X 381.635, Y -281.512, Z 428.603, A 0, B 90, C 0, E1 0, E2 0, E3 0, E4 0}
LIN {X 467.481, Y -275.685, Z 428.605, A 0, B 90, C 0, E1 0, E2 0, E3 0, E4 0}
LIN {X 467.857, Y -280.669, Z 428.762, A 0, B 90, C 0, E1 0, E2 0, E3 0, E4 0}
LIN {X 382.401, Y -286.469, Z 428.76, A 0, B 90, C 0, E1 0, E2 0, E3 0, E4 0}
LIN {X 382.956, Y -291.441, Z 428.917, A 0, B 90, C 0, E1 0, E2 0, E3 0, E4 0}
LIN {X 468.21, Y -285.654, Z 428.919, A 0, B 90, C 0, E1 0, E2 0, E3 0, E4 0}
LIN {X 468.47, Y -290.645, Z 429.076, A 0, B 90, C 0, E1 0, E2 0, E3 0, E4 0}
LIN {X 383.214, Y -296.432, Z 429.074, A 0, B 90, C 0, E1 0, E2 0, E3 0, E4 0}
LIN {X 383.541, Y -301.419, Z 429.23, A 0, B 90, C 0, E1 0, E2 0, E3 0, E4 0}
LIN {X 468.767, Y -295.634, Z 429.232, A 0, B 90, C 0, E1 0, E2 0, E3 0, E4 0}
LIN {X 469.031, Y -300.625, Z 429.389, A 0, B 90, C 0, E1 0, E2 0, E3 0, E4 0}
LIN {X 384.383, Y -306.371, Z 429.387, A 0, B 90, C 0, E1 0, E2 0, E3 0, E4 0}
LIN {X 385.343, Y -311.315, Z 429.544, A 0, B 90, C 0, E1 0, E2 0, E3 0, E4 0}
LIN {X 468.849, Y -305.647, Z 429.546, A 0, B 90, C 0, E1 0, E2 0, E3 0, E4 0}
LIN {X 377.209, Y -261.777, Z 427.976, A 0, B 90, C 0, E1 0, E2 0, E3 0, E4 0}
LIN {X 377.213, Y -261.839, Z 425.977, A 0, B 90, C 0, E1 0, E2 0, E3 0, E4 0}
LIN {X 467.33, Y -255.722, Z 425.979, A 0, B 90, C 0, E1 0, E2 0, E3 0, E4 0}
LIN {X 467.556, Y -260.716, Z 426.136, A 0, B 90, C 0, E1 0, E2 0, E3 0, E4 0}
LIN {X 377.384, Y -266.837, Z 426.134, A 0, B 90, C 0, E1 0, E2 0, E3 0, E4 0}
LIN {X 377.701, Y -271.824, Z 426.29, A 0, B 90, C 0, E1 0, E2 0, E3 0, E4 0}
LIN {X 467.799, Y -265.709, Z 426.293, A 0, B 90, C 0, E1 0, E2 0, E3 0, E4 0}
LIN {X 468.057, Y -270.7, Z 426.449, A 0, B 90, C 0, E1 0, E2 0, E3 0, E4 0}
LIN {X 378.476, Y -276.781, Z 426.447, A 0, B 90, C 0, E1 0, E2 0, E3 0, E4 0}
LIN {X 379.367, Y -281.729, Z 426.604, A 0, B 90, C 0, E1 0, E2 0, E3 0, E4 0}
LIN {X 468.332, Y -275.691, Z 426.606, A 0, B 90, C 0, E1 0, E2 0, E3 0, E4 0}
LIN {X 468.687, Y -280.676, Z 426.763, A 0, B 90, C 0, E1 0, E2 0, E3 0, E4 0}
LIN {X 380.026, Y -286.694, Z 426.761, A 0, B 90, C 0, E1 0, E2 0, E3 0, E4 0}
LIN {X 380.667, Y -291.659, Z 426.918, A 0, B 90, C 0, E1 0, E2 0, E3 0, E4 0}
LIN {X 469.029, Y -285.661, Z 426.92, A 0, B 90, C 0, E1 0, E2 0, E3 0, E4 0}
LIN {X 469.267, Y -290.654, Z 427.076, A 0, B 90, C 0, E1 0, E2 0, E3 0, E4 0}
LIN {X 381.121, Y -296.637, Z 427.074, A 0, B 90, C 0, E1 0, E2 0, E3 0, E4 0}
LIN {X 381.618, Y -301.613, Z 427.231, A 0, B 90, C 0, E1 0, E2 0, E3 0, E4 0}
LIN {X 469.516, Y -295.646, Z 427.233, A 0, B 90, C 0, E1 0, E2 0, E3 0, E4 0}
LIN {X 469.555, Y -300.653, Z 427.39, A 0, B 90, C 0, E1 0, E2 0, E3 0, E4 0}
LIN {X 382.346, Y -306.572, Z 427.388, A 0, B 90, C 0, E1 0, E2 0, E3 0, E4 0}
LIN {X 383.306, Y -311.516, Z 427.545, A 0, B 90, C 0, E1 0, E2 0, E3 0, E4 0}
LIN {X 469.616, Y -305.658, Z 427.547, A 0, B 90, C 0, E1 0, E2 0, E3 0, E4 0}
LIN {X 375.646, Y -261.946, Z 425.977, A 0, B 90, C 0, E1 0, E2 0, E3 0, E4 0}
LIN {X 375.65, Y -262.008, Z 423.978, A 0, B 90, C 0, E1 0, E2 0, E3 0, E4 0}
LIN {X 468.077, Y -255.735, Z 423.98, A 0, B 90, C 0, E1 0, E2 0, E3 0, E4 0}
LIN {X 468.321, Y -260.727, Z 424.137, A 0, B 90, C 0, E1 0, E2 0, E3 0, E4 0}
LIN {X 375.628, Y -267.019, Z 424.134, A 0, B 90, C 0, E1 0, E2 0, E3 0, E4 0}
LIN {X 375.79, Y -272.017, Z 424.291, A 0, B 90, C 0, E1 0, E2 0, E3 0, E4 0}
LIN {X 468.515, Y -265.723, Z 424.293, A 0, B 90, C 0, E1 0, E2 0, E3 0, E4 0}
LIN {X 468.708, Y -270.719, Z 424.45, A 0, B 90, C 0, E1 0, E2 0, E3 0, E4 0}
LIN {X 376.484, Y -276.979, Z 424.448, A 0, B 90, C 0, E1 0, E2 0, E3 0, E4 0}
LIN {X 377.206, Y -281.939, Z 424.605, A 0, B 90, C 0, E1 0, E2 0, E3 0, E4 0}
LIN {X 469.037, Y -275.706, Z 424.607, A 0, B 90, C 0, E1 0, E2 0, E3 0, E4 0}
LIN {X 469.436, Y -280.688, Z 424.764, A 0, B 90, C 0, E1 0, E2 0, E3 0, E4 0}
LIN {X 377.851, Y -286.904, Z 424.762, A 0, B 90, C 0, E1 0, E2 0, E3 0, E4 0}
LIN {X 378.55, Y -291.866, Z 424.918, A 0, B 90, C 0, E1 0, E2 0, E3 0, E4 0}
LIN {X 469.744, Y -285.676, Z 424.921, A 0, B 90, C 0, E1 0, E2 0, E3 0, E4 0}
LIN {X 469.879, Y -290.676, Z 425.077, A 0, B 90, C 0, E1 0, E2 0, E3 0, E4 0}
LIN {X 379.318, Y -296.823, Z 425.075, A 0, B 90, C 0, E1 0, E2 0, E3 0, E4 0}
LIN {X 379.825, Y -301.797, Z 425.232, A 0, B 90, C 0, E1 0, E2 0, E3 0, E4 0}
LIN {X 469.995, Y -295.677, Z 425.234, A 0, B 90, C 0, E1 0, E2 0, E3 0, E4 0}
LIN {X 470.038, Y -300.683, Z 425.391, A 0, B 90, C 0, E1 0, E2 0, E3 0, E4 0}
LIN {X 380.454, Y -306.763, Z 425.389, A 0, B 90, C 0, E1 0, E2 0, E3 0, E4 0}
LIN {X 381.266, Y -311.717, Z 425.546, A 0, B 90, C 0, E1 0, E2 0, E3 0, E4 0}
LIN {X 470.091, Y -305.688, Z 425.548, A 0, B 90, C 0, E1 0, E2 0, E3 0, E4 0}
LIN {X 374.085, Y -262.114, Z 423.978, A 0, B 90, C 0, E1 0, E2 0, E3 0, E4 0}
LIN {X 374.089, Y -262.177, Z 421.979, A 0, B 90, C 0, E1 0, E2 0, E3 0, E4 0}
LIN {X 468.583, Y -255.763, Z 421.981, A 0, B 90, C 0, E1 0, E2 0, E3 0, E4 0}
LIN {X 468.781, Y -260.759, Z 422.138, A 0, B 90, C 0, E1 0, E2 0, E3 0, E4 0}
LIN {X 374.067, Y -267.188, Z 422.135, A 0, B 90, C 0, E1 0, E2 0, E3 0, E4 0}
LIN {X 374.044, Y -272.198, Z 422.292, A 0, B 90, C 0, E1 0, E2 0, E3 0, E4 0}
LIN {X 468.976, Y -265.755, Z 422.294, A 0, B 90, C 0, E1 0, E2 0, E3 0, E4 0}
LIN {X 469.208, Y -270.748, Z 422.451, A 0, B 90, C 0, E1 0, E2 0, E3 0, E4 0}
LIN {X 374.494, Y -277.177, Z 422.449, A 0, B 90, C 0, E1 0, E2 0, E3 0, E4 0}
LIN {X 375.17, Y -282.14, Z 422.606, A 0, B 90, C 0, E1 0, E2 0, E3 0, E4 0}
LIN {X 469.579, Y -275.732, Z 422.608, A 0, B 90, C 0, E1 0, E2 0, E3 0, E4 0}
LIN {X 469.877, Y -280.72, Z 422.765, A 0, B 90, C 0, E1 0, E2 0, E3 0, E4 0}
LIN {X 375.95, Y -287.096, Z 422.763, A 0, B 90, C 0, E1 0, E2 0, E3 0, E4 0}
LIN {X 376.73, Y -292.052, Z 422.919, A 0, B 90, C 0, E1 0, E2 0, E3 0, E4 0}
LIN {X 470.068, Y -285.717, Z 422.921, A 0, B 90, C 0, E1 0, E2 0, E3 0, E4 0}
LIN {X 470.268, Y -290.712, Z 423.078, A 0, B 90, C 0, E1 0, E2 0, E3 0, E4 0}
LIN {X 377.525, Y -297.007, Z 423.076, A 0, B 90, C 0, E1 0, E2 0, E3 0, E4 0}
LIN {X 378.076, Y -301.979, Z 423.233, A 0, B 90, C 0, E1 0, E2 0, E3 0, E4 0}
LIN {X 470.462, Y -295.708, Z 423.235, A 0, B 90, C 0, E1 0, E2 0, E3 0, E4 0}
LIN {X 470.523, Y -300.713, Z 423.392, A 0, B 90, C 0, E1 0, E2 0, E3 0, E4 0}
LIN {X 378.739, Y -306.943, Z 423.39, A 0, B 90, C 0, E1 0, E2 0, E3 0, E4 0}
LIN {X 379.734, Y -311.884, Z 423.547, A 0, B 90, C 0, E1 0, E2 0, E3 0, E4 0}
LIN {X 470.418, Y -305.729, Z 423.549, A 0, B 90, C 0, E1 0, E2 0, E3 0, E4 0}
LIN {X 372.611, Y -262.277, Z 421.978, A 0, B 90, C 0, E1 0, E2 0, E3 0, E4 0}
LIN {X 372.615, Y -262.34, Z 419.979, A 0, B 90, C 0, E1 0, E2 0, E3 0, E4 0}
LIN {X 468.952, Y -255.801, Z 419.982, A 0, B 90, C 0, E1 0, E2 0, E3 0, E4 0}
LIN {X 469.192, Y -260.794, Z 420.138, A 0, B 90, C 0, E1 0, E2 0, E3 0, E4 0}
LIN {X 372.605, Y -267.35, Z 420.136, A 0, B 90, C 0, E1 0, E2 0, E3 0, E4 0}
LIN {X 372.594, Y -272.359, Z 420.293, A 0, B 90, C 0, E1 0, E2 0, E3 0, E4 0}
LIN {X 469.43, Y -265.787, Z 420.295, A 0, B 90, C 0, E1 0, E2 0, E3 0, E4 0}
LIN {X 469.743, Y -270.774, Z 420.452, A 0, B 90, C 0, E1 0, E2 0, E3 0, E4 0}
LIN {X 372.756, Y -277.357, Z 420.45, A 0, B 90, C 0, E1 0, E2 0, E3 0, E4 0}
LIN {X 373.372, Y -282.325, Z 420.607, A 0, B 90, C 0, E1 0, E2 0, E3 0, E4 0}
LIN {X 470.012, Y -275.765, Z 420.609, A 0, B 90, C 0, E1 0, E2 0, E3 0, E4 0}
LIN {X 470.166, Y -280.764, Z 420.766, A 0, B 90, C 0, E1 0, E2 0, E3 0, E4 0}
LIN {X 374.124, Y -287.283, Z 420.763, A 0, B 90, C 0, E1 0, E2 0, E3 0, E4 0}
LIN {X 374.903, Y -292.239, Z 420.92, A 0, B 90, C 0, E1 0, E2 0, E3 0, E4 0}
LIN {X 470.362, Y -285.759, Z 420.922, A 0, B 90, C 0, E1 0, E2 0, E3 0, E4 0}
LIN {X 470.633, Y -290.75, Z 421.079, A 0, B 90, C 0, E1 0, E2 0, E3 0, E4 0}
LIN {X 375.7, Y -297.194, Z 421.077, A 0, B 90, C 0, E1 0, E2 0, E3 0, E4 0}
LIN {X 376.582, Y -302.143, Z 421.234, A 0, B 90, C 0, E1 0, E2 0, E3 0, E4 0}
LIN {X 470.845, Y -295.745, Z 421.236, A 0, B 90, C 0, E1 0, E2 0, E3 0, E4 0}
LIN {X 470.963, Y -300.746, Z 421.393, A 0, B 90, C 0, E1 0, E2 0, E3 0, E4 0}
LIN {X 377.514, Y -307.089, Z 421.391, A 0, B 90, C 0, E1 0, E2 0, E3 0, E4 0}
LIN {X 378.616, Y -312.023, Z 421.547, A 0, B 90, C 0, E1 0, E2 0, E3 0, E4 0}
LIN {X 470.739, Y -305.77, Z 421.55, A 0, B 90, C 0, E1 0, E2 0, E3 0, E4 0}
LIN {X 469.175, Y -255.786, Z 419.982, A 0, B 90, C 0, E1 0, E2 0, E3 0, E4 0}
LIN {X 469.179, Y -255.848, Z 417.983, A 0, B 90, C 0, E1 0, E2 0, E3 0, E4 0}
LIN {X 371.379, Y -262.487, Z 417.98, A 0, B 90, C 0, E1 0, E2 0, E3 0, E4 0}
LIN {X 371.372, Y -267.496, Z 418.137, A 0, B 90, C 0, E1 0, E2 0, E3 0, E4 0}
LIN {X 469.35, Y -260.846, Z 418.139, A 0, B 90, C 0, E1 0, E2 0, E3 0, E4 0}
LIN {X 469.601, Y -265.838, Z 418.296, A 0, B 90, C 0, E1 0, E2 0, E3 0, E4 0}
LIN {X 371.437, Y -272.501, Z 418.294, A 0, B 90, C 0, E1 0, E2 0, E3 0, E4 0}
LIN {X 371.546, Y -277.503, Z 418.451, A 0, B 90, C 0, E1 0, E2 0, E3 0, E4 0}
LIN {X 469.95, Y -270.823, Z 418.453, A 0, B 90, C 0, E1 0, E2 0, E3 0, E4 0}
LIN {X 470.242, Y -275.812, Z 418.61, A 0, B 90, C 0, E1 0, E2 0, E3 0, E4 0}
LIN {X 372.161, Y -282.47, Z 418.607, A 0, B 90, C 0, E1 0, E2 0, E3 0, E4 0}
LIN {X 372.776, Y -287.437, Z 418.764, A 0, B 90, C 0, E1 0, E2 0, E3 0, E4 0}
LIN {X 470.459, Y -280.807, Z 418.767, A 0, B 90, C 0, E1 0, E2 0, E3 0, E4 0}
LIN {X 470.659, Y -285.802, Z 418.923, A 0, B 90, C 0, E1 0, E2 0, E3 0, E4 0}
LIN {X 373.421, Y -292.402, Z 418.921, A 0, B 90, C 0, E1 0, E2 0, E3 0, E4 0}
LIN {X 374.128, Y -297.363, Z 419.078, A 0, B 90, C 0, E1 0, E2 0, E3 0, E4 0}
LIN {X 470.839, Y -290.799, Z 419.08, A 0, B 90, C 0, E1 0, E2 0, E3 0, E4 0}
LIN {X 470.968, Y -295.799, Z 419.237, A 0, B 90, C 0, E1 0, E2 0, E3 0, E4 0}
LIN {X 375.306, Y -302.292, Z 419.235, A 0, B 90, C 0, E1 0, E2 0, E3 0, E4 0}
LIN {X 376.3, Y -307.234, Z 419.392, A 0, B 90, C 0, E1 0, E2 0, E3 0, E4 0}
LIN {X 471.114, Y -300.798, Z 419.394, A 0, B 90, C 0, E1 0, E2 0, E3 0, E4 0}
LIN {X 471.063, Y -305.811, Z 419.55, A 0, B 90, C 0, E1 0, E2 0, E3 0, E4 0}
LIN {X 377.502, Y -312.162, Z 419.548, A 0, B 90, C 0, E1 0, E2 0, E3 0, E4 0}
LIN {X 370.224, Y -262.565, Z 417.98, A 0, B 90, C 0, E1 0, E2 0, E3 0, E4 0}
LIN {X 370.228, Y -262.628, Z 415.981, A 0, B 90, C 0, E1 0, E2 0, E3 0, E4 0}
LIN {X 469.238, Y -255.907, Z 415.984, A 0, B 90, C 0, E1 0, E2 0, E3 0, E4 0}
LIN {X 469.409, Y -260.905, Z 416.14, A 0, B 90, C 0, E1 0, E2 0, E3 0, E4 0}
LIN {X 370.286, Y -267.633, Z 416.138, A 0, B 90, C 0, E1 0, E2 0, E3 0, E4 0}
LIN {X 370.344, Y -272.638, Z 416.295, A 0, B 90, C 0, E1 0, E2 0, E3 0, E4 0}
LIN {X 469.803, Y -265.887, Z 416.297, A 0, B 90, C 0, E1 0, E2 0, E3 0, E4 0}
LIN {X 470.162, Y -270.872, Z 416.454, A 0, B 90, C 0, E1 0, E2 0, E3 0, E4 0}
LIN {X 370.404, Y -277.643, Z 416.452, A 0, B 90, C 0, E1 0, E2 0, E3 0, E4 0}
LIN {X 371.096, Y -282.605, Z 416.608, A 0, B 90, C 0, E1 0, E2 0, E3 0, E4 0}
LIN {X 470.441, Y -275.862, Z 416.611, A 0, B 90, C 0, E1 0, E2 0, E3 0, E4 0}
LIN {X 470.749, Y -280.85, Z 416.767, A 0, B 90, C 0, E1 0, E2 0, E3 0, E4 0}
LIN {X 371.831, Y -287.564, Z 416.765, A 0, B 90, C 0, E1 0, E2 0, E3 0, E4 0}
LIN {X 372.567, Y -292.523, Z 416.922, A 0, B 90, C 0, E1 0, E2 0, E3 0, E4 0}
LIN {X 470.965, Y -285.844, Z 416.924, A 0, B 90, C 0, E1 0, E2 0, E3 0, E4 0}
LIN {X 470.841, Y -290.862, Z 417.081, A 0, B 90, C 0, E1 0, E2 0, E3 0, E4 0}
LIN {X 373.223, Y -297.488, Z 417.079, A 0, B 90, C 0, E1 0, E2 0, E3 0, E4 0}
LIN {X 373.946, Y -302.448, Z 417.236, A 0, B 90, C 0, E1 0, E2 0, E3 0, E4 0}
LIN {X 470.985, Y -295.861, Z 417.238, A 0, B 90, C 0, E1 0, E2 0, E3 0, E4 0}
LIN {X 471.078, Y -300.864, Z 417.395, A 0, B 90, C 0, E1 0, E2 0, E3 0, E4 0}
LIN {X 375.012, Y -307.384, Z 417.392, A 0, B 90, C 0, E1 0, E2 0, E3 0, E4 0}
LIN {X 376.281, Y -312.307, Z 417.549, A 0, B 90, C 0, E1 0, E2 0, E3 0, E4 0}
LIN {X 471.11, Y -305.871, Z 417.551, A 0, B 90, C 0, E1 0, E2 0, E3 0, E4 0}
LIN {X 469.274, Y -255.905, Z 415.984, A 0, B 90, C 0, E1 0, E2 0, E3 0, E4 0}
LIN {X 469.278, Y -255.967, Z 413.985, A 0, B 90, C 0, E1 0, E2 0, E3 0, E4 0}
LIN {X 369.525, Y -262.738, Z 413.982, A 0, B 90, C 0, E1 0, E2 0, E3 0, E4 0}
LIN {X 369.583, Y -267.743, Z 414.139, A 0, B 90, C 0, E1 0, E2 0, E3 0, E4 0}
LIN {X 469.56, Y -260.957, Z 414.141, A 0, B 90, C 0, E1 0, E2 0, E3 0, E4 0}
LIN {X 469.985, Y -265.937, Z 414.298, A 0, B 90, C 0, E1 0, E2 0, E3 0, E4 0}
LIN {X 369.641, Y -272.748, Z 414.296, A 0, B 90, C 0, E1 0, E2 0, E3 0, E4 0}
LIN {X 369.973, Y -277.735, Z 414.453, A 0, B 90, C 0, E1 0, E2 0, E3 0, E4 0}
LIN {X 470.345, Y -270.922, Z 414.455, A 0, B 90, C 0, E1 0, E2 0, E3 0, E4 0}
LIN {X 470.624, Y -275.912, Z 414.612, A 0, B 90, C 0, E1 0, E2 0, E3 0, E4 0}
LIN {X 370.37, Y -282.717, Z 414.61, A 0, B 90, C 0, E1 0, E2 0, E3 0, E4 0}
LIN {X 370.958, Y -287.686, Z 414.766, A 0, B 90, C 0, E1 0, E2 0, E3 0, E4 0}
LIN {X 470.925, Y -280.901, Z 414.769, A 0, B 90, C 0, E1 0, E2 0, E3 0, E4 0}
LIN {X 470.968, Y -285.907, Z 414.925, A 0, B 90, C 0, E1 0, E2 0, E3 0, E4 0}
LIN {X 371.693, Y -292.645, Z 414.923, A 0, B 90, C 0, E1 0, E2 0, E3 0, E4 0}
LIN {X 372.317, Y -297.612, Z 415.08, A 0, B 90, C 0, E1 0, E2 0, E3 0, E4 0}
LIN {X 470.825, Y -290.926, Z 415.082, A 0, B 90, C 0, E1 0, E2 0, E3 0, E4 0}
LIN {X 470.928, Y -295.928, Z 415.239, A 0, B 90, C 0, E1 0, E2 0, E3 0, E4 0}
LIN {X 372.926, Y -302.58, Z 415.237, A 0, B 90, C 0, E1 0, E2 0, E3 0, E4 0}
LIN {X 373.684, Y -307.537, Z 415.394, A 0, B 90, C 0, E1 0, E2 0, E3 0, E4 0}
LIN {X 470.998, Y -300.932, Z 415.396, A 0, B 90, C 0, E1 0, E2 0, E3 0, E4 0}
LIN {X 470.975, Y -305.943, Z 415.553, A 0, B 90, C 0, E1 0, E2 0, E3 0, E4 0}
LIN {X 374.886, Y -312.465, Z 415.55, A 0, B 90, C 0, E1 0, E2 0, E3 0, E4 0}
LIN {X 368.779, Y -262.789, Z 413.983, A 0, B 90, C 0, E1 0, E2 0, E3 0, E4 0}
LIN {X 368.784, Y -262.851, Z 411.984, A 0, B 90, C 0, E1 0, E2 0, E3 0, E4 0}
LIN {X 469.147, Y -256.039, Z 411.986, A 0, B 90, C 0, E1 0, E2 0, E3 0, E4 0}
LIN {X 469.598, Y -261.018, Z 412.143, A 0, B 90, C 0, E1 0, E2 0, E3 0, E4 0}
LIN {X 368.877, Y -267.854, Z 412.14, A 0, B 90, C 0, E1 0, E2 0, E3 0, E4 0}
LIN {X 369.093, Y -272.849, Z 412.297, A 0, B 90, C 0, E1 0, E2 0, E3 0, E4 0}
LIN {X 469.942, Y -266.003, Z 412.299, A 0, B 90, C 0, E1 0, E2 0, E3 0, E4 0}
LIN {X 470.318, Y -270.987, Z 412.456, A 0, B 90, C 0, E1 0, E2 0, E3 0, E4 0}
LIN {X 369.539, Y -277.827, Z 412.454, A 0, B 90, C 0, E1 0, E2 0, E3 0, E4 0}
LIN {X 369.907, Y -282.811, Z 412.611, A 0, B 90, C 0, E1 0, E2 0, E3 0, E4 0}
LIN {X 470.732, Y -275.968, Z 412.613, A 0, B 90, C 0, E1 0, E2 0, E3 0, E4 0}
LIN {X 470.951, Y -280.962, Z 412.77, A 0, B 90, C 0, E1 0, E2 0, E3 0, E4 0}
LIN {X 370.336, Y -287.791, Z 412.767, A 0, B 90, C 0, E1 0, E2 0, E3 0, E4 0}
LIN {X 370.781, Y -292.77, Z 412.924, A 0, B 90, C 0, E1 0, E2 0, E3 0, E4 0}
LIN {X 470.904, Y -285.974, Z 412.927, A 0, B 90, C 0, E1 0, E2 0, E3 0, E4 0}
LIN {X 470.806, Y -290.99, Z 413.083, A 0, B 90, C 0, E1 0, E2 0, E3 0, E4 0}
LIN {X 371.362, Y -297.74, Z 413.081, A 0, B 90, C 0, E1 0, E2 0, E3 0, E4 0}
LIN {X 371.943, Y -302.709, Z 413.238, A 0, B 90, C 0, E1 0, E2 0, E3 0, E4 0}
LIN {X 470.829, Y -295.997, Z 413.24, A 0, B 90, C 0, E1 0, E2 0, E3 0, E4 0}
LIN {X 470.916, Y -301, Z 413.397, A 0, B 90, C 0, E1 0, E2 0, E3 0, E4 0}
LIN {X 372.524, Y -307.679, Z 413.395, A 0, B 90, C 0, E1 0, E2 0, E3 0, E4 0}
LIN {X 373.488, Y -312.622, Z 413.551, A 0, B 90, C 0, E1 0, E2 0, E3 0, E4 0}
LIN {X 470.748, Y -306.021, Z 413.554, A 0, B 90, C 0, E1 0, E2 0, E3 0, E4 0}
PTP {X 430.72, Y -272.354, Z 484.436, A 0, B 90, C 0, E1 0, E2 0, E3 0, E4 0, S 'B010'}
PTP {A1 5, A2 -90, A3 100, A4 5, A5 -10, A6 -5, E1 0, E2 0, E3 0, E4 0} C_PTP

END
